{attribute addProperty BoxType "ATH2000-0250-0022"}
{attribute addProperty Id "A_0014_ATH2050_5501_0022ATH2050_1751249111214"}
{attribute addProperty CRC "489460918"}
{attribute addProperty SizeInBites "112"}
{attribute addProperty SizeInBytes "14"}
TYPE A_0001_ATH2000_0250_0022_1D2C94B6 EXTENDS ATH2000_9506A482 :
STRUCT
	{attribute addProperty Name "A_0014_ATH2050_5501_0022"}
	A_0014_ATH2050_5501_0022 : ATH2050_17512491;
END_STRUCT
END_TYPE

(* stored: Version 1.2.0.0, ProductVersion 3.1.4024.9
   DUT A_0001_ATH2000_0250_0022_1D2C94B6: Id {d92482a0-e018-4fee-96c6-b2c7913b3b95} *)
